TYPE DUT_stOrderItems :
STRUCT
	return_			: DINT;
	BatchId	: STRING(50);
END_STRUCT
END_TYPE

(* stored: Version 1.1.0.1, ProductVersion 3.1.4024.15
   DUT DUT_stOrderItems: Id {c4b8b226-9561-4dee-9759-bfa152eb2ace} *)
